PROGRAM MAIN
VAR
	VarOut AT %Q*: BOOL;
	VarIn AT %I*: BOOL;
END_VAR


VarOut := VarIn;

END_PROGRAM

(* stored: Version 1.1.0.1, ProductVersion 3.1.4024.14
   POU MAIN: Id {9e1b352a-7153-433d-a1b8-938818ae9fd6}, SpecialFunc None *)
